{attribute 'qualified_only'}
{attribute 'strict'}
{attribute 'to_string'}
TYPE DB_COMMAND_DISCONNECTING_STATE :
(
	IDLING,
	DATA_SET_RELEASING,
	DISCONNECTING
);
END_TYPE

(* stored: Version 1.1.0.1
   DUT DB_COMMAND_DISCONNECTING_STATE: Id {04f86573-1447-45fa-af61-017d555b8d41} *)
